// The handle a test body reports through - the object passed as the Test
// parameter of I_Test.Run.
//
// ONE instance per suite, not one per test. Only one test runs at a time, so the
// handle is retargeted to whichever journal is active rather than allocated per
// slot. At capacity 50 that is the difference between one copy of the assertion
// machinery and fifty; the original allocated all of it per slot, which is most of
// why a referencing project paid for it whether it ran tests or not.
//
// Its single job is turning a check into a record: dispatch the comparison,
// compose the diagnostic, count it in the journal and stream it to the detail
// sink. The comparing itself belongs to TestValueCompare, which is pure and
// testable on its own.
//
// Being one per suite is what makes it the right place to hold the detail sink:
// every check in the suite already passes through here, so the sink is one
// reference rather than one per slot.
FUNCTION_BLOCK TestVerdict IMPLEMENTS I_TestAssertions
VAR
	_Journal	: REFERENCE TO TestJournal;
	_DetailSink : I_TestDetailSink;
END_VAR

(*
	No cyclic body. Every entry point is driven by a check in a test body.
*)

// Where individual checks go. Called once by the suite at composition; a null sink
// is the normal case and costs one comparison per check.
//
// Not on I_TestAssertions. A test body holds this object and must not be able to
// redirect the record of its own run.
METHOD AttachDetailSink
VAR_INPUT
	Sink : I_TestDetailSink;
END_VAR
_DetailSink := Sink;
END_METHOD

// Lengths first, so a size difference is reported as one rather than as a
// difference at whatever byte happens to differ.
METHOD AssertBufferEqual
VAR_INPUT
	pExpected	   : POINTER TO BYTE;
	ExpectedLength : UDINT;
	pActual		   : POINTER TO BYTE;
	ActualLength   : UDINT;
	Message		   : T_MaxString;
END_VAR
IF ExpectedLength <> ActualLength THEN
	THIS^.RecordFailure(E_FailureKind.SizeMismatch,
		CONCAT(CONCAT(CONCAT(
		'expected ', LREAL_TO_FMTSTR(TO_LREAL(ExpectedLength), 0, FALSE)),
		' bytes, actual '), LREAL_TO_FMTSTR(TO_LREAL(ActualLength), 0, FALSE)), Message);
	RETURN;
END_IF

THIS^.AssertMemEqual(pExpected, pActual, ExpectedLength, Message);
END_METHOD

// Opt-in, never a default. A scan budget is a real regression signal on a fixed
// target and noise across a matrix of them.
METHOD AssertCompletedWithin
VAR_INPUT
	Cycles	: UDINT;
	Message : T_MaxString;
END_VAR
IF NOT __ISVALIDREF(_Journal) THEN
	RETURN;
END_IF

IF _Journal.ElapsedCycles <= Cycles THEN
	THIS^.RecordPass(Message);
ELSE
	THIS^.RecordFailure(E_FailureKind.Timeout,
		CONCAT(CONCAT(CONCAT(
		'expected within ', LREAL_TO_FMTSTR(TO_LREAL(Cycles), 0, FALSE)),
		' cycles, actual '), LREAL_TO_FMTSTR(TO_LREAL(_Journal.ElapsedCycles), 0, FALSE)),
		Message);
END_IF
END_METHOD

// See TestValueCompare for what equality means here - notably that REAL and
// LREAL compare exactly, and that a size difference is its own failure kind.
METHOD AssertEqual
VAR_INPUT
	Expected : ANY;
	Actual	 : ANY;
	Message	 : T_MaxString;
END_VAR

VAR
	Comparison : ST_CompareResult;
END_VAR
Comparison := TestValueCompare(Expected, Actual);

IF Comparison.IsEqual THEN
	THIS^.RecordPass(Message);
ELSE
	THIS^.Emit(Kind := Comparison.Kind,
			   Expected := Comparison.Expected, Actual := Comparison.Actual,
			   Diagnostic := Comparison.Diagnostic, Message := Message);
END_IF
END_METHOD

METHOD AssertFalse
VAR_INPUT
	Condition : BOOL;
	Message	  : T_MaxString;
END_VAR
IF NOT Condition THEN
	THIS^.RecordPass(Message);
ELSE
	THIS^.RecordFailure(E_FailureKind.ValueMismatch, 'expected FALSE, actual TRUE', Message);
END_IF
END_METHOD

METHOD AssertGreater
VAR_INPUT
	Actual	: ANY;
	Bound	: ANY;
	Message : T_MaxString;
END_VAR

VAR
	ActualNumber : ST_NumericValue;
	BoundNumber	 : ST_NumericValue;
	ExpectedText : T_MaxString;
	ActualText	 : T_MaxString;
END_VAR
ActualNumber := TestValueAsLReal(Actual);
BoundNumber  := TestValueAsLReal(Bound);

IF NOT (ActualNumber.IsNumeric AND BoundNumber.IsNumeric) THEN
	THIS^.RecordFailure(E_FailureKind.TypeMismatch, 'not an ordered type', Message);
ELSIF ActualNumber.Value > BoundNumber.Value THEN
	THIS^.RecordPass(Message);
ELSE
	ExpectedText := CONCAT('greater than ', TestValueString(Bound));
	ActualText	 := TestValueString(Actual);
	THIS^.Emit(Kind := E_FailureKind.ValueMismatch,
			   Expected := ExpectedText, Actual := ActualText,
			   Diagnostic := CONCAT(CONCAT(CONCAT(
					'expected ', TestValueBrief(ExpectedText)),
					', actual '), TestValueBrief(ActualText)),
			   Message := Message);
END_IF
END_METHOD

METHOD AssertInRange
VAR_INPUT
	Actual	: LREAL;
	Minimum : LREAL;
	Maximum : LREAL;
	Message : T_MaxString;
END_VAR
IF (Actual >= Minimum) AND (Actual <= Maximum) THEN
	THIS^.RecordPass(Message);
ELSE
	THIS^.RecordFailure(E_FailureKind.ValueMismatch,
		CONCAT(CONCAT(CONCAT(CONCAT(CONCAT(
		'expected ', LREAL_TO_FMTSTR(Minimum, 6, TRUE)),
		' to '),	 LREAL_TO_FMTSTR(Maximum, 6, TRUE)),
		', actual '), LREAL_TO_FMTSTR(Actual, 6, TRUE)), Message);
END_IF
END_METHOD

PROPERTY AssertionCount : UDINT
GET
IF __ISVALIDREF(_Journal) THEN
	AssertionCount := _Journal.AssertionCount;
END_IF
END_GET
END_PROPERTY

METHOD AssertLess
VAR_INPUT
	Actual	: ANY;
	Bound	: ANY;
	Message : T_MaxString;
END_VAR

VAR
	ActualNumber : ST_NumericValue;
	BoundNumber	 : ST_NumericValue;
	ExpectedText : T_MaxString;
	ActualText	 : T_MaxString;
END_VAR
ActualNumber := TestValueAsLReal(Value := Actual);
BoundNumber  := TestValueAsLReal(Value := Bound);

IF NOT (ActualNumber.IsNumeric AND BoundNumber.IsNumeric) THEN
	THIS^.RecordFailure(E_FailureKind.TypeMismatch, 'not an ordered type', Message);
ELSIF ActualNumber.Value < BoundNumber.Value THEN
	THIS^.RecordPass(Message);
ELSE
	ExpectedText := CONCAT('less than ', TestValueString(Bound));
	ActualText	 := TestValueString(Actual);
	THIS^.Emit(Kind := E_FailureKind.ValueMismatch,
			   Expected := ExpectedText, Actual := ActualText,
			   Diagnostic := CONCAT(CONCAT(CONCAT(
					'expected ', TestValueBrief(ExpectedText)),
					', actual '), TestValueBrief(ActualText)),
			   Message := Message);
END_IF
END_METHOD

METHOD AssertMemEqual
VAR_INPUT
	pExpected : POINTER TO BYTE;
	pActual	  : POINTER TO BYTE;
	Length	  : UDINT;
	Message	  : T_MaxString;
END_VAR

VAR
	pLeft  : POINTER TO BYTE;
	pRight : POINTER TO BYTE;
	i	   : DINT;
END_VAR
IF (pExpected = 0) OR (pActual = 0) THEN
	THIS^.RecordFailure(E_FailureKind.Environment, 'null buffer', Message);
	RETURN;
END_IF

pLeft  := pExpected;
pRight := pActual;

FOR i := 0 TO TO_DINT(Length) - 1 DO
	IF pLeft[i] <> pRight[i] THEN
		THIS^.RecordFailure(E_FailureKind.ValueMismatch,
			CONCAT(CONCAT(CONCAT(CONCAT(CONCAT(
			'differs at byte ', LREAL_TO_FMTSTR(TO_LREAL(i), 0, FALSE)),
			': expected 16#'),	 BYTE_TO_HEXSTR(pLeft[i], 2, TRUE)),
			', actual 16#'),	 BYTE_TO_HEXSTR(pRight[i], 2, TRUE)), Message);
		RETURN;
	END_IF
END_FOR

THIS^.RecordPass(Message);
END_METHOD

// ABSOLUTE tolerance: passes when |Expected - Actual| <= Tolerance.
//
// Tolerance carries the units of the value being compared - millimetres, volts,
// encoder counts. Use it when you know how much error is acceptable in those
// units, which is usually true of a physical measurement.
//
// At large magnitudes an absolute tolerance can fall below what an LREAL can
// represent, at which point it degenerates into exact equality. AssertWithin does
// not have that problem.
METHOD AssertNear
VAR_INPUT
	Expected  : LREAL;
	Actual	  : LREAL;
	Tolerance : LREAL;
	Message	  : T_MaxString;
END_VAR
IF ABS(Expected - Actual) <= ABS(Tolerance) THEN
	THIS^.RecordPass(Message);
ELSE
	THIS^.RecordFailure(E_FailureKind.ValueMismatch,
		CONCAT(CONCAT(CONCAT(CONCAT(CONCAT(
		'expected ', LREAL_TO_FMTSTR(Expected, 6, TRUE)),
		' +/- '),	 LREAL_TO_FMTSTR(ABS(Tolerance), 6, TRUE)),
		', actual '), LREAL_TO_FMTSTR(Actual, 6, TRUE)), Message);
END_IF
END_METHOD

METHOD AssertNotEqual
VAR_INPUT
	Expected : ANY;
	Actual	 : ANY;
	Message	 : T_MaxString;
END_VAR

VAR
	Comparison : ST_CompareResult;
	Rendered   : T_MaxString;
END_VAR
Comparison := TestValueCompare(Expected, Actual);

IF NOT Comparison.IsEqual THEN
	THIS^.RecordPass(Message);
ELSE
	Rendered := TestValueString(Expected);
	THIS^.Emit(Kind := E_FailureKind.ValueMismatch,
			   Expected := CONCAT('any value other than ', Rendered), Actual := Rendered,
			   Diagnostic := CONCAT('expected any value other than ',
									TestValueBrief(Rendered)),
			   Message := Message);
END_IF
END_METHOD

METHOD AssertTrue
VAR_INPUT
	Condition : BOOL;
	Message	  : T_MaxString;
END_VAR
IF Condition THEN
	THIS^.RecordPass(Message);
ELSE
	THIS^.RecordFailure(E_FailureKind.ValueMismatch, 'expected TRUE, actual FALSE', Message);
END_IF
END_METHOD

// RELATIVE tolerance: passes when |Expected - Actual| <= |Expected| * Fraction.
//
// Holds its meaning across magnitudes, which absolute tolerance does not - 0.1 per
// cent means the same thing at 1.0 and at 1E9. Use it for ratios, gains, scaled
// values, and anywhere the acceptable error scales with the value itself.
//
// Near zero it collapses: |Expected| * Fraction approaches nothing, so an expected
// value of zero admits only an exact match. That is not a defect to paper over
// with a hidden floor - if zero is the expected value, an absolute tolerance is
// what the situation calls for, and AssertNear is the method that expresses it.
METHOD AssertWithin
VAR_INPUT
	Expected : LREAL;
	Actual	 : LREAL;

	// Dimensionless. 0.001 is 0.1 per cent of Expected.
	Fraction : LREAL;
	Message	 : T_MaxString;
END_VAR

VAR
	Tolerance : LREAL;
	Detail	  : T_MaxString;
END_VAR
Tolerance := ABS(Expected) * ABS(Fraction);
IF ABS(Expected - Actual) <= Tolerance THEN
	THIS^.RecordPass(Message);
	RETURN;
END_IF

IF Expected = 0.0 THEN
	Detail := CONCAT('expected exactly 0 - a relative tolerance admits nothing else; use AssertNear. Actual ', LREAL_TO_FMTSTR(Actual, 6, TRUE));
	THIS^.RecordFailure(E_FailureKind.ValueMismatch, Detail, Message);
	RETURN;
END_IF

Detail := CONCAT('expected ', LREAL_TO_FMTSTR(Expected, 6, TRUE));
Detail := CONCAT(Detail, ' +/- ');
Detail := CONCAT(Detail, LREAL_TO_FMTSTR(ABS(Fraction) * 100.0, 4, TRUE));
Detail := CONCAT(Detail, '% (');
Detail := CONCAT(Detail, LREAL_TO_FMTSTR(Tolerance, 6, TRUE));
Detail := CONCAT(Detail, '), actual ');
Detail := CONCAT(Detail, LREAL_TO_FMTSTR(Actual, 6, TRUE));
THIS^.RecordFailure(E_FailureKind.ValueMismatch, Detail, Message);
END_METHOD

PROPERTY ElapsedCycles : UDINT
GET
IF __ISVALIDREF(_Journal) THEN
	ElapsedCycles := _Journal.ElapsedCycles;
END_IF
END_GET
END_PROPERTY

PROPERTY ElapsedTime : LREAL
GET
IF __ISVALIDREF(_Journal) THEN
	ElapsedTime := _Journal.ElapsedTime;
END_IF
END_GET
END_PROPERTY

// The one place a failure becomes a record. Private: I_TestOutcome.RecordFailure
// is the public door and delegates here with no values.
//
// Kept private rather than widening RecordFailure because that method is the
// narrow type domain helpers take. An NC helper reporting that an axis never
// homed has no expected-and-actual pair, and should not be made to pass two empty
// strings to say so.
METHOD Emit
VAR_INPUT
	Kind	   : E_FailureKind;
	// Full rendered values, or empty when the failure has no two values.
	Expected   : T_MaxString;
	Actual	   : T_MaxString;
	Diagnostic : T_MaxString;
	Message	   : T_MaxString;
END_VAR

VAR
	StepLabel : T_MaxString;
END_VAR
IF NOT __ISVALIDREF(_Journal) THEN
	RETURN;
END_IF

// The step is read before the journal records anything, so a streamed check
// carries the step it actually ran under.
StepLabel := _Journal.StepLabel;

_Journal.RecordFailure(Kind, Diagnostic, Message);

IF _DetailSink <> 0 THEN
	_DetailSink.CheckFailed(StepLabel := StepLabel, Kind := Kind,
							Expected := Expected, Actual := Actual,
							Diagnostic := Diagnostic, Message := Message);
END_IF
END_METHOD

METHOD Fail
VAR_INPUT
	Reason : T_MaxString;
END_VAR
THIS^.RecordFailure(E_FailureKind.ValueMismatch, 'explicit failure', Reason);
END_METHOD

PROPERTY IsFirstCycle : BOOL
GET
IF __ISVALIDREF(_Journal) THEN
	IsFirstCycle := _Journal.IsFirstCycle;
END_IF
END_GET
END_PROPERTY

METHOD RecordFailure
VAR_INPUT
	Kind	   : E_FailureKind;
	Diagnostic : T_MaxString;
	Message	   : T_MaxString;
END_VAR
THIS^.Emit(Kind := Kind, Expected := '', Actual := '',
		   Diagnostic := Diagnostic, Message := Message);
END_METHOD

METHOD RecordPass
VAR_INPUT
	Detail : T_MaxString;
END_VAR
IF NOT __ISVALIDREF(_Journal) THEN
	RETURN;
END_IF

_Journal.RecordPass();

IF _DetailSink <> 0 THEN
	_DetailSink.CheckPassed(StepLabel := _Journal.StepLabel, Detail := Detail);
END_IF
END_METHOD

METHOD ReportError
VAR_INPUT
	Reason : T_MaxString;
END_VAR
THIS^.RecordFailure(E_FailureKind.Environment, 'could not run', Reason);
END_METHOD

METHOD SetStep
VAR_INPUT
	Label : T_MaxString;
END_VAR
IF __ISVALIDREF(_Journal) THEN
	_Journal.SetStep(Label);
END_IF
END_METHOD

PROPERTY Status : E_TestStatus
GET
IF __ISVALIDREF(_Journal) THEN
	Status := _Journal.Status;
ELSE
	Status := E_TestStatus.NotStarted;
END_IF
END_GET
END_PROPERTY

// Point the handle at nothing. Called by the runner when a test finishes, so a
// stray call cannot write into a completed test's record - or worse, into the
// next test's.
//
// Every method here already guards on __ISVALIDREF, so an untargeted handle is
// inert rather than dangerous. This is what makes that guard mean something.
METHOD Untarget
_Journal REF= 0;
END_METHOD

// Point the handle at the active test's journal. Called by the suite, never by a
// test.
METHOD Target
VAR_INPUT
	Journal : REFERENCE TO TestJournal;
END_VAR
_Journal REF= Journal;
END_METHOD

END_FUNCTION_BLOCK

(* stored: Version 1.1.0.1, ProductVersion 3.1.4026.18
   POU TestVerdict: Id {5110e4c3-37f7-46f6-945d-708582dcd45e}, SpecialFunc None
   Folder I_TestAssertions: Id {e4112d56-62ba-4c84-abb2-d7401a0382bd}
   Folder I_TestOutcome: Id {591f84b0-9ebd-47da-8445-73e8ef5d9a9a}
   Folder I_TestTiming: Id {c05e452e-c8a8-4470-8166-6085e699955a}
   Method AttachDetailSink: Id {95131ad5-92e8-48d6-8c49-0eef69e407db}
   Method AssertBufferEqual: Id {31ca02a3-f5f0-40b4-bb0d-554fb550c585}
   Method AssertCompletedWithin: Id {1f4e4d3b-0ba5-43c1-bad0-bb7c80b0bb38}
   Method AssertEqual: Id {3991bd51-c3f2-4819-bda9-4529a3431716}
   Method AssertFalse: Id {9e4ee1d5-0446-44a2-a24f-7414286d6ca0}
   Method AssertGreater: Id {7d0818f5-774c-4da6-8d94-222e86b766c1}
   Method AssertInRange: Id {f78c48b7-34f7-48d3-9204-2b3e89f6f210}
   Property AssertionCount: Id {6dc42526-bb10-4f7d-baa1-9d3bea6cfeae}
   Get Get: Id {28724282-e36a-4e1e-a885-72d51fc229e1}
   Method AssertLess: Id {a730d242-8c9e-4daf-bf6d-39c8a1e8ff49}
   Method AssertMemEqual: Id {5adc406b-af92-4cc8-a8ac-99e5bb5303d1}
   Method AssertNear: Id {12d11ae7-87cb-4d70-aab5-fc15e3e09ecc}
   Method AssertNotEqual: Id {45468f40-82b0-41ee-86d3-f9f5b13cc0a7}
   Method AssertTrue: Id {9e2c8309-33d4-4304-871a-6df798964fab}
   Method AssertWithin: Id {71a9561c-2e79-4aee-b9f9-e2ffdba558f8}
   Property ElapsedCycles: Id {08b61e99-6795-43f3-b627-cd8467c67f95}
   Get Get: Id {b72f58fb-6e2f-4fcf-8d65-f73904aef68d}
   Property ElapsedTime: Id {6aad5006-fb7a-4415-8a34-d70a7e66d11f}
   Get Get: Id {97166e90-1f91-4a47-b0fe-ee60d2437745}
   Method Emit: Id {07d8a565-131c-4ed3-a08d-a84615a8e145}
   Method Fail: Id {b064e7d8-4cb3-4600-a549-752269d30cc0}
   Property IsFirstCycle: Id {92ba2a3e-d29f-4f99-88bc-881de1e12266}
   Get Get: Id {c7d82c8c-761b-464e-b4d2-5cdfd279b2bb}
   Method RecordFailure: Id {d51ca165-bbc6-44a2-8222-f1836304dc9c}
   Method RecordPass: Id {a1e497db-5d05-4836-8855-da5aac0c1d99}
   Method ReportError: Id {e46b6460-9e55-4a2d-bd66-6440a75e3105}
   Method SetStep: Id {555bdd1a-d4c7-462c-b678-d464d7938840}
   Property Status: Id {8f379328-7f87-4bc8-b315-edc24775da71}
   Get Get: Id {50b31d9b-9378-47c3-bf42-4216abfce6da}
   Method Untarget: Id {c45499c0-5b83-4ad5-b474-dda7b905135f}
   Method Target: Id {3b0923a0-8738-4d87-88fa-9f83fa825da7} *)
